PROGRAM ST_MotionControl
VAR
END_VAR

LD_Y_AXIS_Sagning();

METHOD LD_Y_AXIS_Sagning : BOOL
VAR_INPUT
END_VAR

VAR
END_VAR
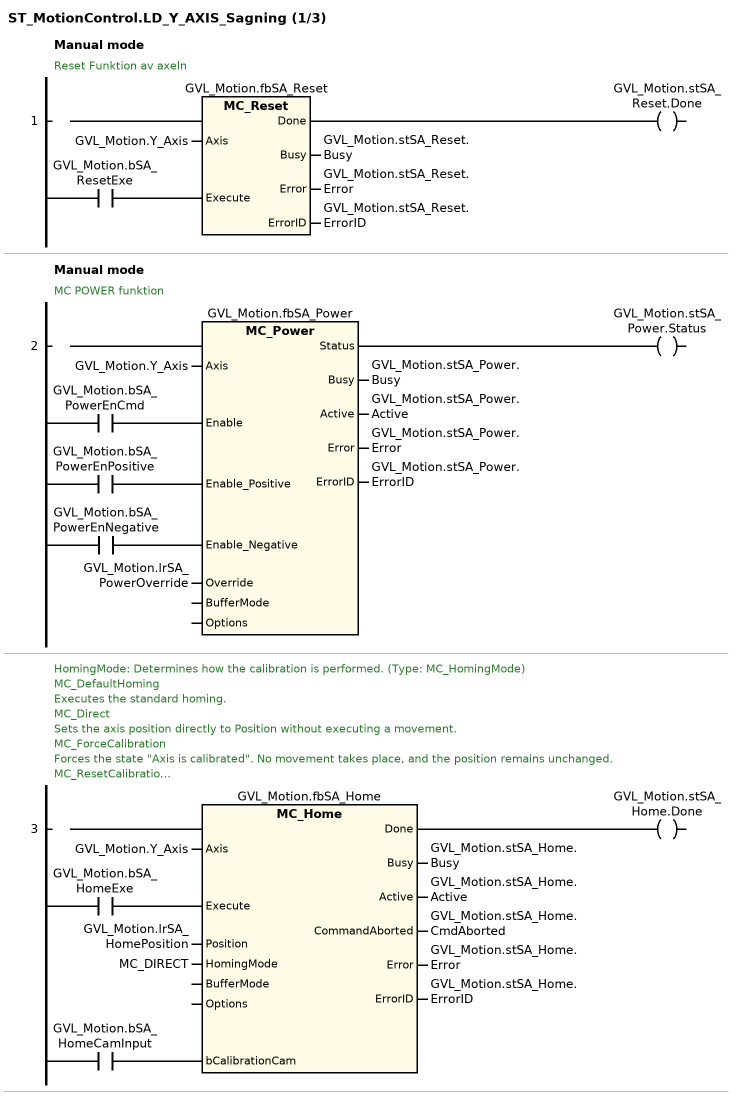
// NETWORK 1: Manual mode
// Reset Funktion av axeln
GVL_Motion.fbSA_Reset(
    Axis := GVL_Motion.Y_Axis,
    Execute := GVL_Motion.bSA_ResetExe,
    Busy => GVL_Motion.stSA_Reset.Busy,
    Error => GVL_Motion.stSA_Reset.Error,
    ErrorID => GVL_Motion.stSA_Reset.ErrorID); // MC_Reset
GVL_Motion.stSA_Reset.Done := GVL_Motion.fbSA_Reset.Done;

// NETWORK 2: Manual mode
// MC POWER funktion
GVL_Motion.fbSA_Power(
    Axis := GVL_Motion.Y_Axis,
    Enable := GVL_Motion.bSA_PowerEnCmd,
    Enable_Positive := GVL_Motion.bSA_PowerEnPositive,
    Enable_Negative := GVL_Motion.bSA_PowerEnNegative,
    Override := GVL_Motion.lrSA_PowerOverride,
    Busy => GVL_Motion.stSA_Power.Busy,
    Active => GVL_Motion.stSA_Power.Active,
    Error => GVL_Motion.stSA_Power.Error,
    ErrorID => GVL_Motion.stSA_Power.ErrorID); // MC_Power
GVL_Motion.stSA_Power.Status := GVL_Motion.fbSA_Power.Status;

// NETWORK 3
// HomingMode: Determines how the calibration is performed. (Type: MC_HomingMode)
//
// MC_DefaultHoming
// Executes the standard homing.
// MC_Direct
// Sets the axis position directly to Position without executing a movement.
// MC_ForceCalibration
// Forces the state "Axis is calibrated". No movement takes place, and the position remains unchanged.
// MC_ResetCalibration
// Resets the calibration status of the axis. No movement takes place, and the position remains unchanged.
// BufferMode: Currently not implemented.
GVL_Motion.fbSA_Home(
    Axis := GVL_Motion.Y_Axis,
    Execute := GVL_Motion.bSA_HomeExe,
    Position := GVL_Motion.lrSA_HomePosition,
    HomingMode := MC_DIRECT,
    bCalibrationCam := GVL_Motion.bSA_HomeCamInput,
    Busy => GVL_Motion.stSA_Home.Busy,
    Active => GVL_Motion.stSA_Home.Active,
    CommandAborted => GVL_Motion.stSA_Home.CmdAborted,
    Error => GVL_Motion.stSA_Home.Error,
    ErrorID => GVL_Motion.stSA_Home.ErrorID); // MC_Home
GVL_Motion.stSA_Home.Done := GVL_Motion.fbSA_Home.Done;

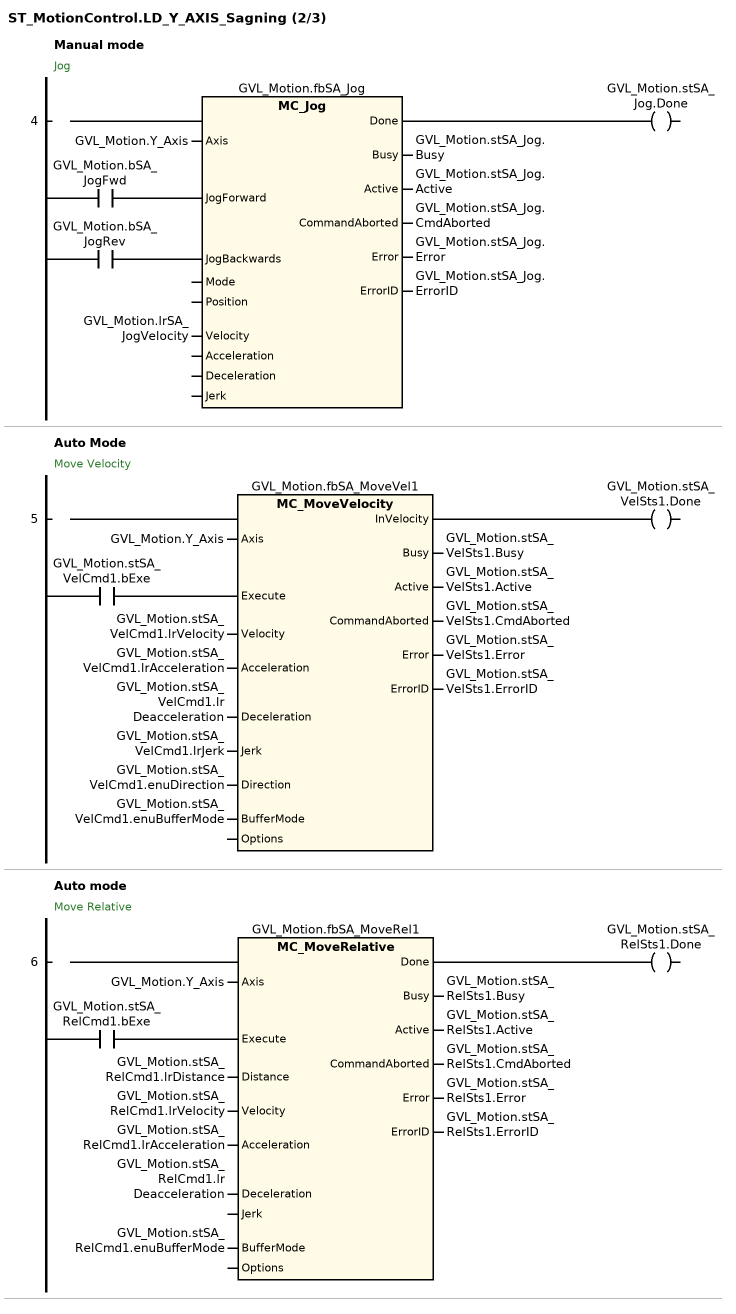
// NETWORK 4: Manual mode
// Jog
GVL_Motion.fbSA_Jog(
    Axis := GVL_Motion.Y_Axis,
    JogForward := GVL_Motion.bSA_JogFwd,
    JogBackwards := GVL_Motion.bSA_JogRev,
    Velocity := GVL_Motion.lrSA_JogVelocity,
    Busy => GVL_Motion.stSA_Jog.Busy,
    Active => GVL_Motion.stSA_Jog.Active,
    CommandAborted => GVL_Motion.stSA_Jog.CmdAborted,
    Error => GVL_Motion.stSA_Jog.Error,
    ErrorID => GVL_Motion.stSA_Jog.ErrorID); // MC_Jog
GVL_Motion.stSA_Jog.Done := GVL_Motion.fbSA_Jog.Done;

// NETWORK 5: Auto Mode
// Move Velocity
GVL_Motion.fbSA_MoveVel1(
    Axis := GVL_Motion.Y_Axis,
    Execute := GVL_Motion.stSA_VelCmd1.bExe,
    Velocity := GVL_Motion.stSA_VelCmd1.lrVelocity,
    Acceleration := GVL_Motion.stSA_VelCmd1.lrAcceleration,
    Deceleration := GVL_Motion.stSA_VelCmd1.lrDeacceleration,
    Jerk := GVL_Motion.stSA_VelCmd1.lrJerk,
    Direction := GVL_Motion.stSA_VelCmd1.enuDirection,
    BufferMode := GVL_Motion.stSA_VelCmd1.enuBufferMode,
    Busy => GVL_Motion.stSA_VelSts1.Busy,
    Active => GVL_Motion.stSA_VelSts1.Active,
    CommandAborted => GVL_Motion.stSA_VelSts1.CmdAborted,
    Error => GVL_Motion.stSA_VelSts1.Error,
    ErrorID => GVL_Motion.stSA_VelSts1.ErrorID); // MC_MoveVelocity
GVL_Motion.stSA_VelSts1.Done := GVL_Motion.fbSA_MoveVel1.InVelocity;

// NETWORK 6: Auto mode
// Move Relative
GVL_Motion.fbSA_MoveRel1(
    Axis := GVL_Motion.Y_Axis,
    Execute := GVL_Motion.stSA_RelCmd1.bExe,
    Distance := GVL_Motion.stSA_RelCmd1.lrDistance,
    Velocity := GVL_Motion.stSA_RelCmd1.lrVelocity,
    Acceleration := GVL_Motion.stSA_RelCmd1.lrAcceleration,
    Deceleration := GVL_Motion.stSA_RelCmd1.lrDeacceleration,
    BufferMode := GVL_Motion.stSA_RelCmd1.enuBufferMode,
    Busy => GVL_Motion.stSA_RelSts1.Busy,
    Active => GVL_Motion.stSA_RelSts1.Active,
    CommandAborted => GVL_Motion.stSA_RelSts1.CmdAborted,
    Error => GVL_Motion.stSA_RelSts1.Error,
    ErrorID => GVL_Motion.stSA_RelSts1.ErrorID); // MC_MoveRelative
GVL_Motion.stSA_RelSts1.Done := GVL_Motion.fbSA_MoveRel1.Done;

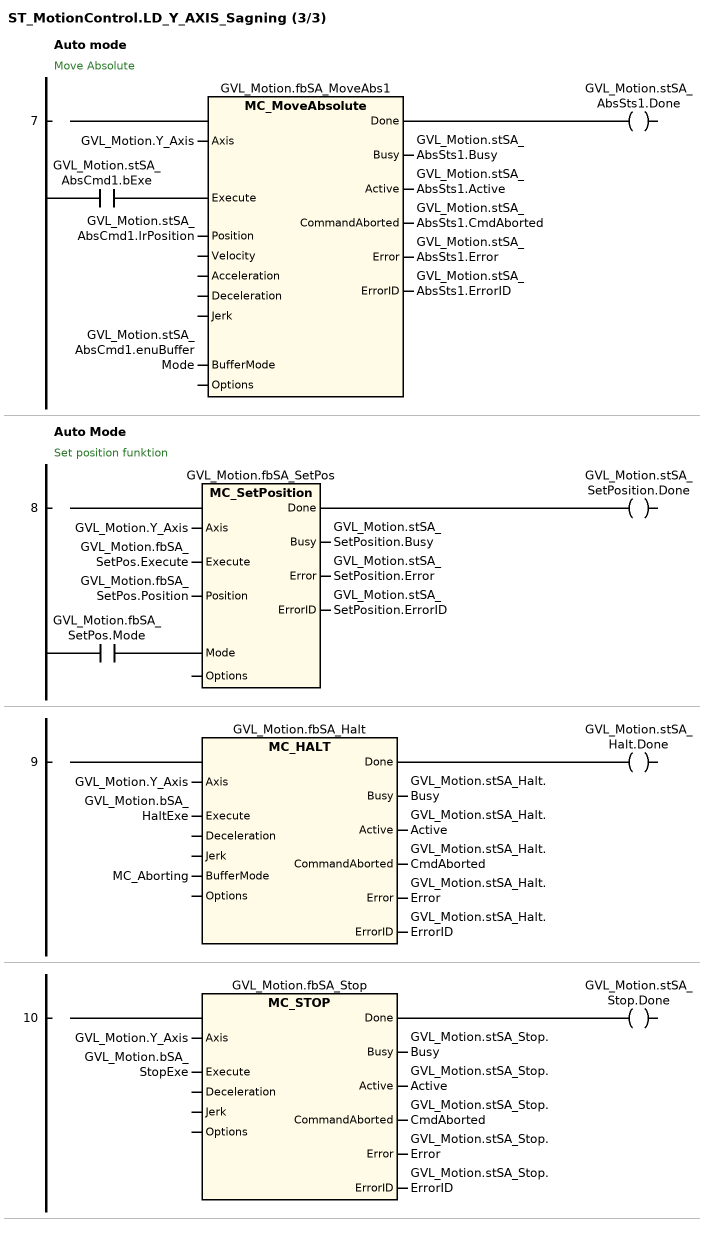
// NETWORK 7: Auto mode
// Move Absolute
GVL_Motion.fbSA_MoveAbs1(
    Axis := GVL_Motion.Y_Axis,
    Execute := GVL_Motion.stSA_AbsCmd1.bExe,
    Position := GVL_Motion.stSA_AbsCmd1.lrPosition,
    BufferMode := GVL_Motion.stSA_AbsCmd1.enuBufferMode,
    Busy => GVL_Motion.stSA_AbsSts1.Busy,
    Active => GVL_Motion.stSA_AbsSts1.Active,
    CommandAborted => GVL_Motion.stSA_AbsSts1.CmdAborted,
    Error => GVL_Motion.stSA_AbsSts1.Error,
    ErrorID => GVL_Motion.stSA_AbsSts1.ErrorID); // MC_MoveAbsolute
GVL_Motion.stSA_AbsSts1.Done := GVL_Motion.fbSA_MoveAbs1.Done;

// NETWORK 8: Auto Mode
// Set position funktion
GVL_Motion.fbSA_SetPos(
    Axis := GVL_Motion.Y_Axis,
    Execute := GVL_Motion.fbSA_SetPos.Execute,
    Position := GVL_Motion.fbSA_SetPos.Position,
    Mode := GVL_Motion.fbSA_SetPos.Mode,
    Busy => GVL_Motion.stSA_SetPosition.Busy,
    Error => GVL_Motion.stSA_SetPosition.Error,
    ErrorID => GVL_Motion.stSA_SetPosition.ErrorID); // MC_SetPosition
GVL_Motion.stSA_SetPosition.Done := GVL_Motion.fbSA_SetPos.Done;

// NETWORK 9
GVL_Motion.fbSA_Halt(
    Axis := GVL_Motion.Y_Axis,
    Execute := GVL_Motion.bSA_HaltExe,
    BufferMode := MC_Aborting,
    Busy => GVL_Motion.stSA_Halt.Busy,
    Active => GVL_Motion.stSA_Halt.Active,
    CommandAborted => GVL_Motion.stSA_Halt.CmdAborted,
    Error => GVL_Motion.stSA_Halt.Error,
    ErrorID => GVL_Motion.stSA_Halt.ErrorID); // MC_HALT
GVL_Motion.stSA_Halt.Done := GVL_Motion.fbSA_Halt.Done;

// NETWORK 10
GVL_Motion.fbSA_Stop(
    Axis := GVL_Motion.Y_Axis,
    Execute := GVL_Motion.bSA_StopExe,
    Busy => GVL_Motion.stSA_Stop.Busy,
    Active => GVL_Motion.stSA_Stop.Active,
    CommandAborted => GVL_Motion.stSA_Stop.CmdAborted,
    Error => GVL_Motion.stSA_Stop.Error,
    ErrorID => GVL_Motion.stSA_Stop.ErrorID); // MC_STOP
GVL_Motion.stSA_Stop.Done := GVL_Motion.fbSA_Stop.Done;
END_METHOD

END_PROGRAM

(* stored: Version 1.1.0.1, ProductVersion 3.1.4024.10
   POU ST_MotionControl: Id {41bc2555-b157-40f0-a097-c1767125ae2b}, SpecialFunc None
   Method LD_Y_AXIS_Sagning: Id {7bba080a-35d2-4745-9c96-d52f0a3d7d43} *)
